{attribute 'qualified_only'}
{attribute 'strict'}
TYPE ParallelModes :
(
	Unknown := 0, Idle, Standalone, Slave, Master
);
END_TYPE

(* stored: Version 1.1.0.1, ProductVersion 3.1.4024.6
   DUT ParallelModes: Id {8e1c2d79-6e46-4358-bedf-dbcb07d9ea82} *)
